{attribute 'qualified_only'}
{attribute 'strict'}
TYPE E_Mode :
(
	AUTO := 0,
	OFF := 1,
	MANUAL := 2
);
END_TYPE

(* stored: Version 1.1.0.1, ProductVersion 3.1.4024.12
   DUT E_Mode: Id {232568a8-6914-43b5-a613-832433836990} *)
